// TIA Portal V19 export
DATA_BLOCK "Measurement_Data"   // DB2
{ S7_Optimized_Access := 'FALSE' }
   VAR RETAIN
      Length : Real;
      Last_Measurement : Real;
      Encoder_Cnt : DInt;
      Pulses_Per_Meter : DInt := 2048;
      Reset : Bool;
      Data_Logger_Bit : Bool;
   END_VAR
BEGIN
END_DATA_BLOCK
